(* IEC 61131-3 sources: CodesysTest/alpha/export/Pro18_1174_04.dev/Plc Logic/Application/Motors/Applied Motion/FB_AppliedMotionStepServoMBBase.pou, 1 file *)

(* ---- ExecuteStoredProgram.m.st ---- *)
(*#-#-#-#-#-#-#-#-#-#---Declaration---#-#-#-#-#-#-#-#-#-#-#-#-#*)

METHOD ExecuteStoredProgram
VAR_INPUT
    (*Program number to execute*)
    programNumber    : INT;
END_VAR
(*#-#-#-#-#-#-#-#-#-#---Implementation---#-#-#-#-#-#-#-#-#-#-#-#-#*)
